# EPICS autosave request: iocBoot/sioc-esb-bkh8/bkh8.req
file ../bkhAnalI.req P=$(P),MOD=3162-$(M),N=1
file ../bkhAnalI.req P=$(P),MOD=3162-$(M),N=2

file ../bkhAnalI.req P=$(P),MOD=3064-$(M),N=1
file ../bkhAnalI.req P=$(P),MOD=3064-$(M),N=2
file ../bkhAnalI.req P=$(P),MOD=3064-$(M),N=3
file ../bkhAnalI.req P=$(P),MOD=3064-$(M),N=4

file ../bkhAnalI.req P=$(P),MOD=3314C-$(M),N=1
file ../bkhAnalI.req P=$(P),MOD=3314C-$(M),N=2
file ../bkhAnalI.req P=$(P),MOD=3314C-$(M),N=3
file ../bkhAnalI.req P=$(P),MOD=3314C-$(M),N=4
file ../bkhAnalI.req P=$(P),MOD=3314C-$(M),N=5
file ../bkhAnalI.req P=$(P),MOD=3314C-$(M),N=6
file ../bkhAnalI.req P=$(P),MOD=3314C-$(M),N=7
file ../bkhAnalI.req P=$(P),MOD=3314C-$(M),N=8

file ../bkhAnalI.req P=$(P),MOD=3314F-$(M),N=1
file ../bkhAnalI.req P=$(P),MOD=3314F-$(M),N=2
file ../bkhAnalI.req P=$(P),MOD=3314F-$(M),N=3
file ../bkhAnalI.req P=$(P),MOD=3314F-$(M),N=4
file ../bkhAnalI.req P=$(P),MOD=3314F-$(M),N=5
file ../bkhAnalI.req P=$(P),MOD=3314F-$(M),N=6
file ../bkhAnalI.req P=$(P),MOD=3314F-$(M),N=7
file ../bkhAnalI.req P=$(P),MOD=3314F-$(M),N=8

file ../bkhDigiO.req P=$(P),MOD=2114-$(M),N=1
file ../bkhDigiO.req P=$(P),MOD=2114-$(M),N=2
file ../bkhDigiO.req P=$(P),MOD=2114-$(M),N=3
file ../bkhDigiO.req P=$(P),MOD=2114-$(M),N=4
file ../bkhDigiO.req P=$(P),MOD=2114-$(M),N=5
file ../bkhDigiO.req P=$(P),MOD=2114-$(M),N=6
file ../bkhDigiO.req P=$(P),MOD=2114-$(M),N=7
file ../bkhDigiO.req P=$(P),MOD=2114-$(M),N=8

file ../bkhDigiO.req P=$(P),MOD=2124-$(M),N=1
file ../bkhDigiO.req P=$(P),MOD=2124-$(M),N=2
file ../bkhDigiO.req P=$(P),MOD=2124-$(M),N=3
file ../bkhDigiO.req P=$(P),MOD=2124-$(M),N=4
file ../bkhDigiO.req P=$(P),MOD=2124-$(M),N=5
file ../bkhDigiO.req P=$(P),MOD=2124-$(M),N=6
file ../bkhDigiO.req P=$(P),MOD=2124-$(M),N=7
file ../bkhDigiO.req P=$(P),MOD=2124-$(M),N=8

file ../bkhDigiI.req P=$(P),MOD=1124-$(M),N=1
file ../bkhDigiI.req P=$(P),MOD=1124-$(M),N=2
file ../bkhDigiI.req P=$(P),MOD=1124-$(M),N=3
file ../bkhDigiI.req P=$(P),MOD=1124-$(M),N=4
